// TIA Portal V17 export
// export: Created 2025-03-07T09:19:07.8643394Z, ExportSetting WithDefaults, DisplayName Totally Integrated Automation Portal, DisplayVersion V17 Update 8, DisplayName TIA Portal Openness, DisplayVersion V17 Update 8, DisplayName TIA Portal Version Control Interface, DisplayVersion V17, DisplayName SINAMICS Startdrive Advanced, DisplayVersion V17 SP2, DisplayName SINAMICS Startdrive G110M, G120, G120C, G120D, G120P, G115D, DisplayVersion V17 SP2, DisplayName SINAMICS Startdrive G130, G150, S120, S150, SINAMICS MV, S210, DisplayVersion V17 SP2, DisplayName STEP 7 Professional, DisplayVersion V17 Update 8, DisplayName SINUMERIK ONE STEP 7 Toolbox, DisplayVersion V17 Update 12, DisplayName SINUMERIK 840D sl STEP 7 Toolbox, DisplayVersion V17 Update 12, DisplayName STEP 7 Safety, DisplayVersion V17 Update 6, DisplayName WinCC Advanced, DisplayVersion V17 Update 8
FUNCTION "FC10200_PYROMETERS" : Void   // FC10200, LAD
{ S7_Optimized_Access := 'TRUE' }
VERSION : 0.1
// stored: AutoNumber false, IsIECCheckEnabled false, SetENOAutomatically false, UDAEnableTagReadback false
BEGIN

REGION Network 1: /////_UNIT_01_/////
END_REGION

REGION Network 2: SENSOR INPUTS
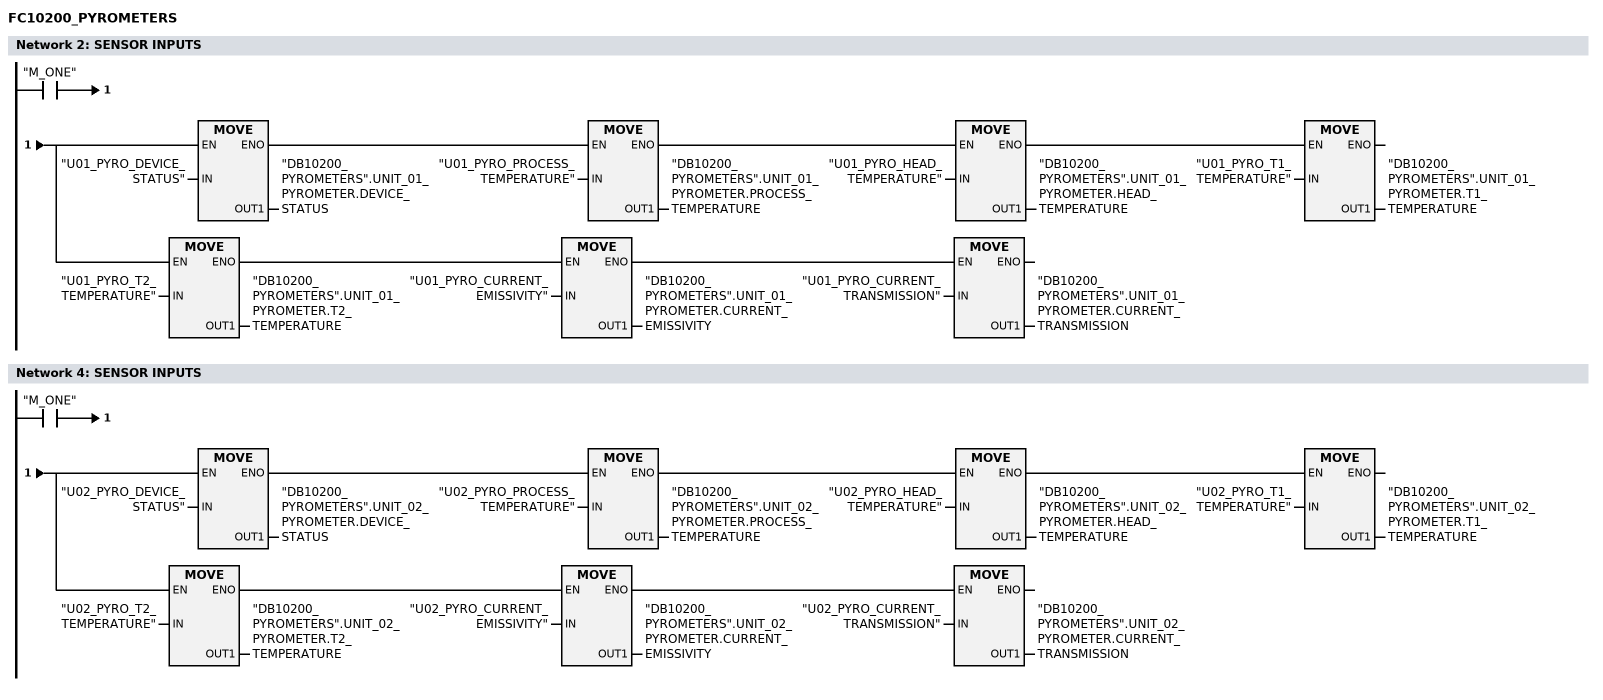
   RUNG wire#powerrail
      Contact( "M_ONE" )
      wire#w1
      Move(in := "U01_PYRO_DEVICE_STATUS", out1 => "DB10200_PYROMETERS".UNIT_01_PYROMETER.DEVICE_STATUS)
      Move(in := "U01_PYRO_PROCESS_TEMPERATURE", out1 => "DB10200_PYROMETERS".UNIT_01_PYROMETER.PROCESS_TEMPERATURE)
      Move(in := "U01_PYRO_HEAD_TEMPERATURE", out1 => "DB10200_PYROMETERS".UNIT_01_PYROMETER.HEAD_TEMPERATURE)
      Move(in := "U01_PYRO_T1_TEMPERATURE", out1 => "DB10200_PYROMETERS".UNIT_01_PYROMETER.T1_TEMPERATURE)
   END_RUNG
   RUNG wire#w1
      Move(in := "U01_PYRO_T2_TEMPERATURE", out1 => "DB10200_PYROMETERS".UNIT_01_PYROMETER.T2_TEMPERATURE)
      Move(in := "U01_PYRO_CURRENT_EMISSIVITY", out1 => "DB10200_PYROMETERS".UNIT_01_PYROMETER.CURRENT_EMISSIVITY)
      Move(in := "U01_PYRO_CURRENT_TRANSMISSION", out1 => "DB10200_PYROMETERS".UNIT_01_PYROMETER.CURRENT_TRANSMISSION)
   END_RUNG
   // the same network as SCL:
   IF "M_ONE" THEN
       "DB10200_PYROMETERS".UNIT_01_PYROMETER.DEVICE_STATUS := "U01_PYRO_DEVICE_STATUS";
       "DB10200_PYROMETERS".UNIT_01_PYROMETER.PROCESS_TEMPERATURE := "U01_PYRO_PROCESS_TEMPERATURE";
       "DB10200_PYROMETERS".UNIT_01_PYROMETER.HEAD_TEMPERATURE := "U01_PYRO_HEAD_TEMPERATURE";
       "DB10200_PYROMETERS".UNIT_01_PYROMETER.T1_TEMPERATURE := "U01_PYRO_T1_TEMPERATURE";
       "DB10200_PYROMETERS".UNIT_01_PYROMETER.T2_TEMPERATURE := "U01_PYRO_T2_TEMPERATURE";
       "DB10200_PYROMETERS".UNIT_01_PYROMETER.CURRENT_EMISSIVITY := "U01_PYRO_CURRENT_EMISSIVITY";
       "DB10200_PYROMETERS".UNIT_01_PYROMETER.CURRENT_TRANSMISSION := "U01_PYRO_CURRENT_TRANSMISSION";
   END_IF;
END_REGION

REGION Network 3: /////_UNIT_02_/////
END_REGION

REGION Network 4: SENSOR INPUTS
   RUNG wire#powerrail
      Contact( "M_ONE" )
      wire#w1
      Move(in := "U02_PYRO_DEVICE_STATUS", out1 => "DB10200_PYROMETERS".UNIT_02_PYROMETER.DEVICE_STATUS)
      Move(in := "U02_PYRO_PROCESS_TEMPERATURE", out1 => "DB10200_PYROMETERS".UNIT_02_PYROMETER.PROCESS_TEMPERATURE)
      Move(in := "U02_PYRO_HEAD_TEMPERATURE", out1 => "DB10200_PYROMETERS".UNIT_02_PYROMETER.HEAD_TEMPERATURE)
      Move(in := "U02_PYRO_T1_TEMPERATURE", out1 => "DB10200_PYROMETERS".UNIT_02_PYROMETER.T1_TEMPERATURE)
   END_RUNG
   RUNG wire#w1
      Move(in := "U02_PYRO_T2_TEMPERATURE", out1 => "DB10200_PYROMETERS".UNIT_02_PYROMETER.T2_TEMPERATURE)
      Move(in := "U02_PYRO_CURRENT_EMISSIVITY", out1 => "DB10200_PYROMETERS".UNIT_02_PYROMETER.CURRENT_EMISSIVITY)
      Move(in := "U02_PYRO_CURRENT_TRANSMISSION", out1 => "DB10200_PYROMETERS".UNIT_02_PYROMETER.CURRENT_TRANSMISSION)
   END_RUNG
   // the same network as SCL:
   IF "M_ONE" THEN
       "DB10200_PYROMETERS".UNIT_02_PYROMETER.DEVICE_STATUS := "U02_PYRO_DEVICE_STATUS";
       "DB10200_PYROMETERS".UNIT_02_PYROMETER.PROCESS_TEMPERATURE := "U02_PYRO_PROCESS_TEMPERATURE";
       "DB10200_PYROMETERS".UNIT_02_PYROMETER.HEAD_TEMPERATURE := "U02_PYRO_HEAD_TEMPERATURE";
       "DB10200_PYROMETERS".UNIT_02_PYROMETER.T1_TEMPERATURE := "U02_PYRO_T1_TEMPERATURE";
       "DB10200_PYROMETERS".UNIT_02_PYROMETER.T2_TEMPERATURE := "U02_PYRO_T2_TEMPERATURE";
       "DB10200_PYROMETERS".UNIT_02_PYROMETER.CURRENT_EMISSIVITY := "U02_PYRO_CURRENT_EMISSIVITY";
       "DB10200_PYROMETERS".UNIT_02_PYROMETER.CURRENT_TRANSMISSION := "U02_PYRO_CURRENT_TRANSMISSION";
   END_IF;
END_REGION
END_FUNCTION
